PROGRAM MAIN
VAR
	bSwitchCtrl		: BOOL := TRUE;
	nRotateUpper	: WORD := 16#8000;
	nRotateLower	: WORD := 16#01;
	
	//Variables for dynamically changing the devices spoken to over EtherCAT
	uiSlaveAddr : UINT;
	nDriveNum	: BYTE;
	nDriveType	: BYTE;
	//For the sake of demonstration I am going to employ a CASE switch for talking to the various drives when initializing...
	iNumDrives	: UINT := 1;
	iDriveType	: UINT := 123;
	
	//Hardware inputs
	bEL1004_CH4 AT%I*	: BOOL;
	stPlcDriveRef AT %I* : ST_PlcDriveRef;
	
	
	nEL2008_value AT%Q*	: BYTE;
	//Comms Retry Timer
	tRetryComms		: TON;
	bTimerDone		: BOOL;
	
	//Booleans for circulating the comms for the drives 
	bInit1 : BOOL := FALSE;
	bInit2 : BOOL := FALSE;
	bInit3 : BOOL := FALSE;
	bInit4 : BOOL := FALSE;
	
	//Log the amount of times the communications have failed:
	iDriveCommsFailure1 : INT := 0;
	iDriveCommsFailure2 : INT := 0;
	iDriveCommsFailure3 : INT := 0;
	iDriveCommsFailure4 : INT := 0;
	
	//Booleans for capturing drive failures
	bBadDriveComms1 : BOOL := FALSE;
	bBadDriveComms2 : BOOL := FALSE;
	bBadDriveComms3 : BOOL := FALSE;
	bBadDriveComms4 : BOOL := FALSE;
	
	//bHaltCommRetries
	aHaltCommsRetries : ARRAY[0..iNumDrives] OF BOOL;
	i : UINT; // for use in the for loop
	bDoHaltCommsInitOnce : BOOL := FALSE;
	bCommsError : BOOL := FALSE;
	bHoldAllComms : BOOL := FALSE;
	
	//Function Block references
	fbWriteCommandControl 	: FB_SoEWriteCommandControl_ByDriveRef;
	bWriteCommand			: BOOL;	
	
	//Exception Handling Variables
	exception 		: __SYSTEM.ExceptionCode;
	lastException 	: __SYSTEM.ExceptionCode;
	pSample			: POINTER TO BOOL;
	bVar			: BOOL;
	nSample			: INT := 100;
	nDivisor		: INT;
	iNumDrives_CATCH	: INT;

	
END_VAR

VAR_INPUT
	//Reference to the drive. The reference to the drive can be linked directly to the PLC in the System Manager. 
	//To do this, an instance of the structure ST_PlcDriveRef must be allocated and the NetID must be converted from the byte array into a string. (Type: ST_DriveRef)
	stDriveRef	: ST_DriveRef;
	//Parameter number to which fbWriteCommandControl refers, e.g. "P_0_IDN + 23" for P-0-0023
	nIdn		: WORD;
	//Indicates, if a command should be prepared (eSoE_CmdControl_Set := 1), executed (eSoE_CmdControl_SetAndEnable := 3) or aborted (eSoE_CmdControl_Cancel := 0).
	eCmdControl	: E_SoE_CmdControl;
	//The function block is enabled via a positive edge at this input
	bExecute	: BOOL;
	//Maximum time (10 s) allowed for the execution of the function block.
	tTimeout	: TIME := DEFAULT_ADS_TIMEOUT;	
END_VAR

VAR_OUTPUT
	//This output is set when the function block is activated, and remains set until a feedback is received.
	bBusy			: BOOL;
	//This output is set after the bBusy output has been reset when an error occurs in the transmission of the command.
	bError			: BOOL;
	//In the case of a set bError output returns the ADS error code of the last executed command.
	iAdsErrId		: UINT;
	//In the case of a set bError output returns the Sercos error of the last executed command.
	iSercosErrId	: UINT;
END_VAR

(*This portion is for dynamic drive communication*)

(*Drives have to be made contact with initially before anything can continue...*)
//Start of the array values for use in the comms logic
IF NOT bDoHaltCommsInitOnce THEN
FOR i := 0 TO iNumDrives DO
	aHaltCommsRetries[i] := FALSE;
END_FOR
	bDoHaltCommsInitOnce := TRUE;
END_IF

//Loop through the comms to determine if any error occurs...
IF NOT bHoldAllComms THEN
FOR i := 0 TO iNumDrives DO
bCommsError := aHaltCommsRetries[i] = TRUE;
IF bCommsError THEN
	bHoldAllComms := TRUE;
END_IF
END_FOR
END_IF

IF NOT bHoldAllComms THEN
// A __TRY __CATCH __FINALLY clause will be added for exception handling shortly...
CASE iNumDrives OF //probably the conditional control function I like the most...
//Setting up comms for the motion control needs
	1: 	__TRY	
	
		IF NOT bInit1 AND NOT aHaltCommsRetries[iNumDrives] THEN

			//change the Slave address
			uiSlaveAddr := iNumDrives;
			GVL_VAR.uiSlaveAddr := uiSlaveAddr;
			//The structure created for the ST_DriveRef expects a Byte format...hence the conversion of the ints...
			GVL_VAR.nDriveNum	:= INT_TO_BYTE(iNumDrives);
			GVL_VAR.nDriveType	:= INT_TO_BYTE(iDriveType);

			stDriveRef.sNetId		:=	F_CreateAmsNetId(stPlcDriveRef.aNetId);
			//The following values have been preconfigured by the FB
			stDriveRef.nSlaveAddr	:=	GVL_VAR.uiSlaveAddr;
			stDriveRef.nDriveNo		:=	GVL_VAR.nDriveNum;
			stDriveRef.nDriveType	:=	GVL_VAR.nDriveType;
	
		IF (stDriveRef.sNetId <> '') AND (stDriveRef.nSlaveAddr <> 0) THEN
		
			bInit1 := TRUE;//initialization completed
		
		END_IF
		END_IF
		
		IF bWriteCommand AND bInit1 THEN
	
			fbWriteCommandControl(
				stDriveRef	:= stDriveRef,
				bExecute	:= TRUE,
				tTimeout	:= DEFAULT_ADS_TIMEOUT,//possible ADSLOGSTR correlation (ADS)
				nIdn		:= P_0_IDN + 23,
				eCmdControl := eCmdControl
				);
		IF NOT	fbWriteCommandControl.bBusy THEN
			fbWriteCommandControl(stDriveRef := stDriveRef, bExecute := FALSE);
			bWriteCommand := FALSE;			
		END_IF
		END_IF
	
		__CATCH(exception)//the variable 'exception' is used to store the error code
	
			iNumDrives_CATCH	:= iNumDrives_CATCH +1;
			F_SaveExceptionCode.excInput := exception;
			iDriveCommsFailure1 := UINT_TO_INT(iNumDrives);
			bBadDriveComms1 := TRUE;

		__FINALLY // The __FINALLY clause will always execute irrespective of the previous commands' success
			
			//If the value that is stored is ever to become TRUE, the code may not be run again
			aHaltCommsRetries[iNumDrives] := iDriveCommsFailure1 = 5;
			//increment for the next case...
		IF	NOT bBadDriveComms1 AND iDriveCommsFailure1 < 5 THEN
			iNumDrives := iNumDrives + 1;
			iDriveCommsFailure1 := 0;
			
			
		ELSE
			//Add in a retry clause for the sake of establishing comms after initial error
			tRetryComms(IN := TRUE, PT:=T#500MS, Q=> btimerDone);
		IF tRetryComms.Q THEN
			//reinitialize the first drive comms attempt
			bInit1 := FALSE; 
			iNumDrives := 1;
			tRetryComms.IN := FALSE;		
		END_IF
		END_IF
	
 		__ENDTRY
		
	2:	__TRY

		IF NOT bInit2 THEN
	
			//change the Slave address
			uiSlaveAddr := iNumDrives;
			GVL_VAR.uiSlaveAddr := uiSlaveAddr;
			//The structure created for the ST_DriveRef expects a Byte format...hence the conversion of the ints...
			GVL_VAR.nDriveNum	:= INT_TO_BYTE(iNumDrives);
			GVL_VAR.nDriveType	:= INT_TO_BYTE(iDriveType);

			stDriveRef.sNetId		:=	F_CreateAmsNetId(stPlcDriveRef.aNetId);
			//The following values have been preconfigured by the FB
			stDriveRef.nSlaveAddr	:=	GVL_VAR.uiSlaveAddr;
			stDriveRef.nDriveNo		:=	GVL_VAR.nDriveNum;
			stDriveRef.nDriveType	:=	GVL_VAR.nDriveType;
	
		IF (stDriveRef.sNetId <> '') AND (stDriveRef.nSlaveAddr <> 0) THEN
		
			bInit2 := TRUE;//initialization completed
		
		END_IF
	
		END_IF
		
		IF bWriteCommand AND bInit2 THEN
	
			fbWriteCommandControl(
				stDriveRef	:= stDriveRef,
				bExecute	:= TRUE,
				tTimeout	:= DEFAULT_ADS_TIMEOUT,
				nIdn		:= P_0_IDN + 23,
				eCmdControl := eCmdControl
				);
		IF NOT	fbWriteCommandControl.bBusy THEN
			fbWriteCommandControl(stDriveRef := stDriveRef, bExecute := FALSE);
			bWriteCommand := FALSE;			
		END_IF
		END_IF
		
		__CATCH(exception)//the variable 'exception' is used to store the error code
	
			iNumDrives_CATCH	:= iNumDrives_CATCH +1;
			F_SaveExceptionCode.excInput := exception;
			iDriveCommsFailure2 := UINT_TO_INT(iNumDrives);
			bBadDriveComms2 := TRUE;

		__FINALLY // The __FINALLY clause will always execute irrespective of the previous commands' success

				//increment for the next case...
		IF	NOT bBadDriveComms2 AND iDriveCommsFailure2 < 5 THEN
			iNumDrives := iNumDrives + 1;
			iDriveCommsFailure2 := 0;
		ELSE
			//Add in a retry clause for the sake of establishing comms after initial error
			tRetryComms(IN := TRUE, PT:=T#500MS, Q=> btimerDone);
		IF tRetryComms.Q THEN
			//reinitialize the first drive comms attempt
			bInit2 := FALSE; 
			iNumDrives := 2;
			tRetryComms.IN := FALSE;		
		END_IF
		END_IF
	
 		__ENDTRY
		
		
	
	3:	__TRY

		IF NOT bInit3 THEN
	
			//change the Slave address
			uiSlaveAddr := iNumDrives;
			GVL_VAR.uiSlaveAddr := uiSlaveAddr;
			//The structure created for the ST_DriveRef expects a Byte format...hence the conversion of the ints...
			GVL_VAR.nDriveNum	:= INT_TO_BYTE(iNumDrives);
			GVL_VAR.nDriveType	:= INT_TO_BYTE(iDriveType);

			stDriveRef.sNetId		:=	F_CreateAmsNetId(stPlcDriveRef.aNetId);
			//The following values have been preconfigured by the FB
			stDriveRef.nSlaveAddr	:=	GVL_VAR.uiSlaveAddr;
			stDriveRef.nDriveNo		:=	GVL_VAR.nDriveNum;
			stDriveRef.nDriveType	:=	GVL_VAR.nDriveType;
	
		IF (stDriveRef.sNetId <> '') AND (stDriveRef.nSlaveAddr <> 0) THEN
		
			bInit3 := TRUE;//initialization completed
		
		END_IF
	
		END_IF
		
		IF bWriteCommand AND bInit3 THEN
	
			fbWriteCommandControl(
				stDriveRef	:= stDriveRef,
				bExecute	:= TRUE,
				tTimeout	:= DEFAULT_ADS_TIMEOUT,
				nIdn		:= P_0_IDN + 23,
				eCmdControl := eCmdControl
				);
		IF NOT	fbWriteCommandControl.bBusy THEN
			fbWriteCommandControl(stDriveRef := stDriveRef, bExecute := FALSE);
			bWriteCommand := FALSE;			
		END_IF
		END_IF

		__CATCH(exception)//the variable 'exception' is used to store the error code
	
			iNumDrives_CATCH	:= iNumDrives_CATCH +1;
			F_SaveExceptionCode.excInput := exception;
			iDriveCommsFailure3 := UINT_TO_INT(iNumDrives);
			bBadDriveComms3 := TRUE;

		__FINALLY // The __FINALLY clause will always execute irrespective of the previous commands' success

				//increment for the next case...
		IF	NOT bBadDriveComms3 AND iDriveCommsFailure3 < 5 THEN
			iNumDrives := iNumDrives + 1;
			iDriveCommsFailure1 := 0;
		ELSE
			//Add in a retry clause for the sake of establishing comms after initial error
			tRetryComms(IN := TRUE, PT:=T#500MS, Q=> btimerDone);
		IF tRetryComms.Q THEN
			//reinitialize the first drive comms attempt
			bInit3 := FALSE; 
			iNumDrives := 3;
			tRetryComms.IN := FALSE;		
		END_IF
		END_IF
	
 		__ENDTRY
		

	
	4:	__TRY

		IF NOT bInit4 THEN
	
		//change the Slave address
		uiSlaveAddr := iNumDrives;
		GVL_VAR.uiSlaveAddr := uiSlaveAddr;
		//The structure created for the ST_DriveRef expects a Byte format...hence the conversion of the ints...
		GVL_VAR.nDriveNum	:= INT_TO_BYTE(iNumDrives);
		GVL_VAR.nDriveType	:= INT_TO_BYTE(iDriveType);

		stDriveRef.sNetId		:=	F_CreateAmsNetId(stPlcDriveRef.aNetId);
		//The following values have been preconfigured by the FB
		stDriveRef.nSlaveAddr	:=	GVL_VAR.uiSlaveAddr;
		stDriveRef.nDriveNo		:=	GVL_VAR.nDriveNum;
		stDriveRef.nDriveType	:=	GVL_VAR.nDriveType;
	
		IF (stDriveRef.sNetId <> '') AND (stDriveRef.nSlaveAddr <> 0) THEN
		
		bInit4 := TRUE;//initialization completed
		
		END_IF
	
		END_IF
		
		IF bWriteCommand AND bInit4 THEN
	
			fbWriteCommandControl(
				stDriveRef	:= stDriveRef,
				bExecute	:= TRUE,
				tTimeout	:= DEFAULT_ADS_TIMEOUT,
				nIdn		:= P_0_IDN + 23,
				eCmdControl := eCmdControl
				);
		IF NOT	fbWriteCommandControl.bBusy THEN
			fbWriteCommandControl(stDriveRef := stDriveRef, bExecute := FALSE);
			bWriteCommand := FALSE;			
		END_IF	
		END_IF

		__CATCH(exception)//the variable 'exception' is used to store the error code
	
			iNumDrives_CATCH	:= iNumDrives_CATCH +1;
			F_SaveExceptionCode.excInput := exception;
			iDriveCommsFailure4 := UINT_TO_INT(iNumDrives);
			bBadDriveComms4 := TRUE;

		__FINALLY // The __FINALLY clause will always execute irrespective of the previous commands' success

				//increment for the next case...
		IF	NOT bBadDriveComms4 AND iDriveCommsFailure4 < 5 THEN
			iNumDrives := iNumDrives + 1;
			iDriveCommsFailure4 := 0;
		ELSE
			//Add in a retry clause for the sake of establishing comms after initial error
			tRetryComms(IN := TRUE, PT:=T#500MS, Q=> btimerDone);
		IF tRetryComms.Q THEN
			//reinitialize the first drive comms attempt
			bInit4 := FALSE; 
			iNumDrives := 4;
			tRetryComms.IN := FALSE;		
		END_IF
		END_IF
	
 		__ENDTRY

END_CASE
END_IF



IF bEL1004_CH4 THEN
	IF bSwitchCtrl THEN
		bSwitchCtrl := FALSE;
		nRotateLower := ROL(nRotateUpper, 2);
		nRotateUpper := ROR(nRotateUpper, 2);
		nEL2008_value := WORD_TO_BYTE(nRotateLower OR nRotateUpper);
	END_IF
ELSE
		IF NOT bSwitchCtrl THEN
			bSwitchCtrl := TRUE;
		END_IF
END_IF

END_PROGRAM

(* stored: Version 1.1.0.1, ProductVersion 3.1.4024.12
   POU MAIN: Id {61722ceb-acc8-4a94-a17e-a2b60d2331d1}, SpecialFunc None *)
